% RSLogix 500 project math block.RSS, saved by version 8.30.00.15 %
PROJECT "UNTITLED"    % processor: MicroLogix 1000 %

PROGRAM FILES
  LAD 2 "MAIN_PROG"  6 rungs
  LAD 3 "USER_FAULT"  1 rungs
  LAD 4 "HSC_INT"  1 rungs
  LAD 5 "STI_INT"  1 rungs
  LAD 6, 7, 8, 9, 10, 11, 12, 13, 14, 15, 16: only END

DATA FILES
  O0 OUTPUT  1 elements
  I1 INPUT  2 elements
  S2 STATUS  33 elements
  B3 BINARY  32 elements
  T4 TIMER  40 elements
  C5 COUNTER  32 elements
  R6 CONTROL  16 elements
  N7 INTEGER  105 elements

LADDER 2 "MAIN_PROG"
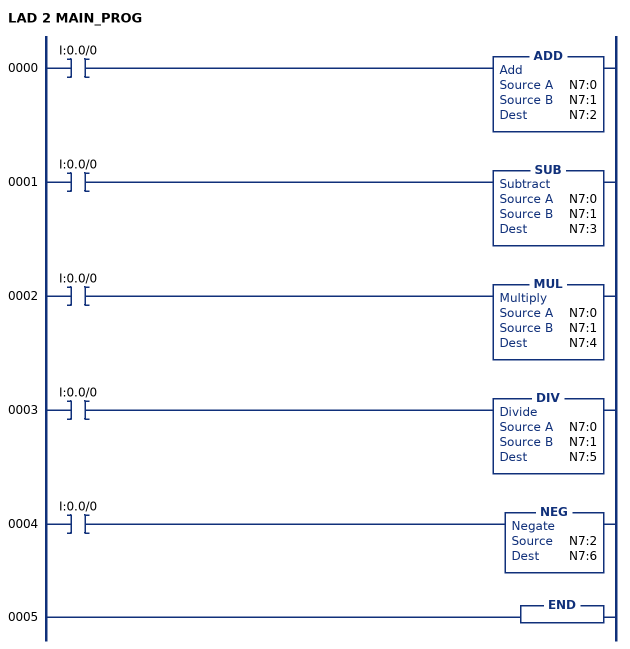
% Rung: 0 %
SOR XIC I:0.0/0 ADD N7:0 N7:1 N7:2 EOR
% Rung: 1 %
SOR XIC I:0.0/0 SUB N7:0 N7:1 N7:3 EOR
% Rung: 2 %
SOR XIC I:0.0/0 MUL N7:0 N7:1 N7:4 EOR
% Rung: 3 %
SOR XIC I:0.0/0 DIV N7:0 N7:1 N7:5 EOR
% Rung: 4 %
SOR XIC I:0.0/0 NEG N7:2 N7:6 EOR
% Rung: 5 %
SOR END EOR

DATA TABLE (non-zero values as saved)
DATA N7
% N7:0 % 10 5 15 5 50 2 -15 0 0 0
